(* CODESYS project PFC200_SMS_Alarm.project
   Company: Storm Elektro

Project tree, tasks and I/O mapping:
  PFC200_2ETH_RS_3G : 750-8217 PFC200, WAGO, order no. 750-8217, version 6.1.0.17
    application Application
      libraries: Standard, 3.5.18.0 (System); WagoAppPlcModbus, 1.1.4.8 (WAGO); WagoAppDatalogger, 1.0.5.3 (WAGO); VisuDialogs, * (System); CmpBitmapPool, * (System)
      task Task (cyclic, interval t#50ms, priority 15) calls alarm_test
      task VISU_TASK (cyclic, interval 100 ms, priority 15) calls VisuElems.Visu_Prg
      Symbols
      global variables PersistentVars
      global variables GVL_SMS
      data type DUT_alarm
      text list AlarmListe
      visualisation Visualization
      program alarm_test [ST]: ACT_alarmtekst, ACT_AlarmGruppe, ACT_Alarmliste, ACT_AlarmMottakere, ACT_ReceivdSMS, ACT_SMS_Tjenesten, ACT_ST_SMS_test, ACT_MappingIO
      image pool ImagePool
    Kbus : Kbus, WAGO, version 2.1.0.1
        unmapped channels: K-BUS diagnostics
      XZ200 : 750-1405, WAGO, order no. 750-1405, version 2.0.0.14
          input  xInput1 : BOOL  // _IN._IN
          input  xInput2 : BOOL  // _IN._IN
          input  xInput3 : BOOL  // _IN._IN
          input  xInput4 : BOOL  // _IN._IN
          input  xInput5 : BOOL  // _IN._IN
          input  xInput6 : BOOL  // _IN._IN
          input  xInput7 : BOOL  // _IN._IN
          input  xInput8 : BOOL  // _IN._IN
          input  xInput9 : BOOL  // _IN._IN
          input  xInput10 : BOOL  // _IN._IN
          input  xInput11 : BOOL  // _IN._IN
          input  xInput12 : BOOL  // _IN._IN
          input  xInput13 : BOOL  // _IN._IN
          input  xInput14 : BOOL  // _IN._IN
          input  xInput15 : BOOL  // _IN._IN
          input  xInput16 : BOOL  // _IN._IN
          unmapped channels: _IN
      XZ201 : 750-1405, WAGO, order no. 750-1405, version 2.0.0.14
          input  xInput17 : BOOL  // _IN._IN
          input  xInput18 : BOOL  // _IN._IN
          input  xInput19 : BOOL  // _IN._IN
          input  xInput20 : BOOL  // _IN._IN
          input  xInput21 : BOOL  // _IN._IN
          input  xInput22 : BOOL  // _IN._IN
          input  xInput23 : BOOL  // _IN._IN
          input  xInput24 : BOOL  // _IN._IN
          input  xInput25 : BOOL  // _IN._IN
          input  xInput26 : BOOL  // _IN._IN
          input  xInput27 : BOOL  // _IN._IN
          input  xInput28 : BOOL  // _IN._IN
          input  xInput29 : BOOL  // _IN._IN
          input  xInput30 : BOOL  // _IN._IN
          input  xInput31 : BOOL  // _IN._IN
          input  xInput32 : BOOL  // _IN._IN
          unmapped channels: _IN
      XZ202 : 750-1405, WAGO, order no. 750-1405, version 2.0.0.14
          input  xInput33 : BOOL  // _IN._IN
          input  xInput34 : BOOL  // _IN._IN
          input  xInput35 : BOOL  // _IN._IN
          input  xInput36 : BOOL  // _IN._IN
          input  xInput37 : BOOL  // _IN._IN
          input  xInput38 : BOOL  // _IN._IN
          input  xInput39 : BOOL  // _IN._IN
          input  xInput40 : BOOL  // _IN._IN
          input  xInput41 : BOOL  // _IN._IN
          input  xInput42 : BOOL  // _IN._IN
          input  xInput43 : BOOL  // _IN._IN
          input  xInput44 : BOOL  // _IN._IN
          input  xInput45 : BOOL  // _IN._IN
          input  xInput46 : BOOL  // _IN._IN
          input  xInput47 : BOOL  // _IN._IN
          input  xInput48 : BOOL  // _IN._IN
          unmapped channels: _IN
    Serial
      COM1 : COM1, WAGO, version 0.0.0.19
  libraries: WagoAppSerial_Sms, 1.6.3.2 (WAGO); VisuSymbols, 4.1.0.0 (System); WagoVisuIcons, 1.1.0.5 (WAGO); WagoVisuIconsMaterialDesign, 1.0.0.0 (WAGO)
  text list GlobalTextList
  5ce3da45-db07-42e7-a21c-a00fff4ed8f6|C:\Users\esbo\Downloads\stormlogo.png
*)

// PFC200_2ETH_RS_3G/Application/DUT_alarm
TYPE DUT_alarm :
STRUCT
	TP_Alarm		    : TP;				// Trigger på alarmer
	tTid			    : TIME := T#1S;		// tid
	xAlarm			    : BOOL;				// Alarmgrupper Alarmer som er der nå.
    xAlarm_Trigger      : BOOL;             // Trigger Alarm for å telle antall alarmer
	xIO_input		    : BOOL;				// Input for alarm before timer, enable,disable
	xEnable			    : BOOL := TRUE;		// Enable alarm
	rTrig_Alarm		    : R_TRIG;
	iAlarm_Aktive	    : INT := 0;         // Teller opp antall aktive alarmer
    iAlarm_Ukvitterte	: INT := 0;         // Teller opp antall alarmer siden sist kvittering.
	sAlarmgruppe	    : STRING(255);
	sPrioritet		    : STRING(2);
    xAlarm_GUI          : BOOL;             // alarm til gui
END_STRUCT
END_TYPE

// PFC200_2ETH_RS_3G/Application/PersistentVars
{attribute 'qualified_only'}
VAR_GLOBAL PERSISTENT RETAIN

END_VAR

// PFC200_2ETH_RS_3G/Application/GVL_SMS
{attribute 'qualified_only'}
VAR_GLOBAL
	sAlarmgruppe		: STRING;		// Melding om hvilke alarmgruppe som er utløst
	iAlarmerAktive		: INT := 0;
    iAlarm_Ukvitterte	: INT := 0;         // Teller opp antall alarmer siden sist kvittering.

    xAlarm_GUI          : BOOL;             // alarm til gui
	iAlarmerSendtSMS	: INT := 0;
	iNull				: INT := 0;


	// Trigger SMS sending fra Alarmgruppe, henter det opp i AlarmMottakere 
	xTriggerSms: BOOL;
	// Reseter tellere iAlarmerAktive og iAlarmerSendt
	xKvitter				: BOOL;
	sKvitteringsord			: STRING := 'Kvittert';	//Kvitterings ord
	sKvittering				: STRING := 'Alarmer er kvittert';	//Kvitterings ord
	
	// SMS test
	sSMStest				: STRING := 'Dette er en test av sms sending';	//Kvitterings ord
	xSMStest				: BOOL;	// Test sending av sms
	
END_VAR

VAR_GLOBAL RETAIN
	xNewSmsReceived			: BOOL;
	sMessage				: STRING(GSM_SMS_MSG_MAX_LENGTH);
	// Klargjort for at det skal sendes SMS hvis xTriggerSms og xMobilNR er TRUE
	xMobil_Send				: BOOL;
	xMobil_1_Send			: BOOL;
	xMobil_2_Send			: BOOL;
	xMobil_3_Send			: BOOL;
	iSignalQuality			: INT; 
	xError					: BOOL;    
	oStatus					: WagoSysErrorBase.FbResult;     
	
(*-------------- Melding som skal sendes til SMS Tjeneste ---------------------*)
	xNyMelding				: BOOL := FALSE;
	sNyMelding				: STRING;		// Melding som skal sendes til SMS Tjenesten
	// Alarmvarsel!
	sAlarmVarsel			: STRING(255) := 'Alarm! ' ;
	// AlarmSted
	sAlarmSted				: STRING(255) := 'Alarm place';
	sPrioritet		        : STRING(2);
(*-------------------------------------------------------------------------------------------------------*)
	// Oppdatere mobilNR
	xMobilNR1_CMD			: BOOL := TRUE;
	sMobilNR1				: STRING := '12345678' ;
    xMobilNR1_A_CMD			: BOOL := TRUE;
    xMobilNR1_B_CMD			: BOOL := TRUE; 
    
	xMobilNR2_CMD			: BOOL := TRUE;
	sMobilNR2				: STRING := '87654321' ;
    xMobilNR2_A_CMD			: BOOL := TRUE;
    xMobilNR2_B_CMD			: BOOL := FALSE;     
    
	xMobilNR3_CMD			: BOOL := TRUE;
	sMobilNR3				: STRING := '56784321' ;
    xMobilNR3_A_CMD			: BOOL := TRUE;
    xMobilNR3_B_CMD			: BOOL := TRUE; 
(*--------------Forsinkelse hvis man ikke får kvitterings sms før ny sms sendes---------------------*)
	// Forsinkelsestid
	tAlarmForsinkelse		: TIME := T#24H ;
(*-------------- Pin kode --------------------------------------------------------------------------*)
sPin				: STRING := '9999';	(*pin1: for your sim card like ‘1234’. Empty String means -> no Pin needed*) 

END_VAR

// PFC200_2ETH_RS_3G/Application/alarm_test
PROGRAM alarm_test
VAR
(*----------------------------------------- SMS BLOKK ------------------------------------------------------*)	
(*FbSimpleSms_8207_0	: FbSimpleSms_8207;*)
(*Modem 				: WagoTypesCom.I_WagoSysComBase;*)

my_utSms                 : WagoSysModem.typRxSms;


//xTxInternational	: BOOL;     
my_sTxMessage			: STRING(SMS_CONSTANT.SMS_MSG_MAX_LENGTH) := 'Hello fra SMS_sending' ;			(*(GSM_SMS_MSG_MAX_LENGTH)*) 
my_sTxNumber			: STRING(SMS_CONSTANT.SMS_MSG_MAX_LENGTH) := '12881288';			(*(GSM_PHONE_NO_MAX_LENGTH)*)     
my_receivedMsg          : STRING(SMS_CONSTANT.SMS_MSG_MAX_LENGTH);
my_xTxTriggerSms		: BOOL;				(*start transmission *)
typMy_receivedMsg       : typDeliverSms;
oModemStatus            : WagoSysErrorBase.FbResult;
xSmsSend                : BOOL;				(*TRUE signals that a new message was received -> the application have TO reset THIS variable*) 


GsmMessage              : typGsmMessage;
RxSms                   : typRxSms;
StatusSms               : typStatusSms;
TimeStamp               : typTimeStamp;
UserDataHeader          : typUserDataHeader;

// utTypRxSms 			: wagoappserial_sms.typRxSms;			(*received sms*) 
// eLastSendState		: eErrorGsm;		(*eErrorGsm.OK*)   
//eLastSendStateOK	: eErrorGsm := OK;
// iTxMsgRefNo			: INT; 
(*-------------------------------------------------------------------------------------------------------*)	

	(*--------------Varaibler til FOR LOOP alarmer---------------------*)
	iNull			: INT := 0;
	i				: INT := 0;
	aAlarm			: ARRAY[1..50] OF DUT_alarm;
    iAlarmerAktive_Temp		: INT := 0;
    iAlarm_Ukvitterte_Temp	: INT := 0;         // Teller opp antall alarmer siden sist kvittering.
    
    (*--------------Variabler til GUI------------------------------------*)
	j				: INT := 1;
    k				: INT := 2;
    l				: INT := 3;
    wJ              : WORD := 1;
    dwFillColorAL   : DWORD := 16#FFFF0000;
    dwFrameColorAL   : DWORD := 16#FFFF0000;
    xTest           : BOOL;
    
	(*--------------Forsinkelse hvis man ikke får kvitterings sms før ny sms sendes---------------------*)
	AlarmTimer				: TON;			//Forsinkelse før jeg sender ny alarm
	tAlarmTidCurrent		: TIME;
	xAlarmTidStart			: BOOL;			// Start timer
END_VAR

ACT_alarmtekst();	// Overfører data fra alarm til array

ACT_AlarmGruppe();

ACT_Alarmliste();

ACT_AlarmMottakere();

ACT_SMS_Tjenesten();
ACT_ReceivdSMS();
ACT_ST_SMS_test();
ACT_MappingIO();




//  --- Send SMS
Modem.SmsSend(  sSMSC_No   :='', 
                sDest_No   := my_sTxNumber,
                sMessage   := my_receivedMsg,
                xTxTrigger := my_xTxTriggerSms,
                oStatus    => oModemStatus,
            );


// GUI program
k := j + 1;
l := k + 1;

j := WORD_TO_INT(wJ);

GVL_SMS.xAlarm_GUI := (GVL_SMS.iAlarmerAktive > 0);

ACTION ACT_alarmtekst:
aAlarm[1].sAlarmgruppe := 'B-Alarm Lav temperatur sprinklertank 1';
aAlarm[2].sAlarmgruppe := 'B-Alarm Lav temperatur sprinklertank 2';
aAlarm[3].sAlarmgruppe := 'B-Alarm SM017 ventil stengt';
aAlarm[4].sAlarmgruppe := 'B-Alarm SM015-SM016 ventil stengt';
aAlarm[5].sAlarmgruppe := 'B-Alarm SM010 ventil stengt';
aAlarm[6].sAlarmgruppe := 'B-Alarm SM013-SM014 ventil stengt';
aAlarm[7].sAlarmgruppe := 'B-Alarm SM019 ventil stengt';
aAlarm[8].sAlarmgruppe := 'B-Alarm SM021 ventil stengt'; 
aAlarm[9].sAlarmgruppe := 'B-Alarm SM022 ventil stengt';
aAlarm[10].sAlarmgruppe := 'B-Alarm SM023 ventil stengt';
aAlarm[11].sAlarmgruppe := 'B-Alarm SM024 ventil stengt';
aAlarm[12].sAlarmgruppe := 'B-Alarm SM003-SM004 ventil stengt';
aAlarm[13].sAlarmgruppe := 'B-Alarm QP001 lavt trykk kommunal ledning';
aAlarm[14].sAlarmgruppe := 'B-Alarm SM001-SM002 ventil stengt';
aAlarm[15].sAlarmgruppe := 'B-Alarm SM025 ventil stengt';
aAlarm[16].sAlarmgruppe := 'B-Alarm RT001 lav temperatur pumperom';

aAlarm[17].sAlarmgruppe := 'B-Alarm Sprinklerpumpe 1 - i drift';
aAlarm[18].sAlarmgruppe := 'B-Alarm Sprinklerpumpe 1 - Motor alarm';
aAlarm[19].sAlarmgruppe := 'B-Alarm Sprinklerpumpe 1 - Automatikk alarm';
aAlarm[20].sAlarmgruppe := 'B-Alarm Sprinklerpumpe 1 – Pumperom alarm';
aAlarm[21].sAlarmgruppe := 'B-Alarm Sprinklerpumpe 1 – Ikke i Auto';
aAlarm[22].sAlarmgruppe := 'B-Alarm SM012 ventil stengt';
aAlarm[23].sAlarmgruppe := 'B-Alarm RN003 Lavt nivå sprinklertank 1';
aAlarm[24].sAlarmgruppe := 'B-Alarm RN004 Høy nivå sprinklertank 1';
aAlarm[25].sAlarmgruppe := 'B-Alarm Sprinklerpumpe 2 - i drift';
aAlarm[26].sAlarmgruppe := 'B-Alarm Sprinklerpumpe 2 - Motor alarm';
aAlarm[27].sAlarmgruppe := 'B-Alarm Sprinklerpumpe 2 - Automatikk alarm';
aAlarm[28].sAlarmgruppe := 'B-Alarm Sprinklerpumpe 2 – Pumperom alarm';
aAlarm[29].sAlarmgruppe := 'B-Alarm Sprinklerpumpe 2 – Ikke i Auto';
aAlarm[30].sAlarmgruppe := 'B-Alarm RN005 Lavt nivå sprinklertank 2';
aAlarm[31].sAlarmgruppe := 'A-Alarm RN006 Høy nivå sprinklertank 2';
aAlarm[32].sAlarmgruppe := 'Ledig';
aAlarm[33].sAlarmgruppe := 'A-Alarm Sprinkler utløst pumperom';
aAlarm[34].sAlarmgruppe := 'A-Alarm Sprinklerpumpe 1 i drift';
aAlarm[35].sAlarmgruppe := 'A-Alarm Sprinklerpumpe 2 i drift';

aAlarm[1].sPrioritet := 'B';
aAlarm[2].sPrioritet := 'B';
aAlarm[3].sPrioritet := 'B';
aAlarm[4].sPrioritet := 'B';
aAlarm[5].sPrioritet := 'B';
aAlarm[6].sPrioritet := 'B';
aAlarm[7].sPrioritet := 'B';
aAlarm[8].sPrioritet := 'B';
aAlarm[9].sPrioritet := 'B';
aAlarm[10].sPrioritet := 'B';
aAlarm[11].sPrioritet := 'B';
aAlarm[12].sPrioritet := 'B';
aAlarm[13].sPrioritet := 'B';
aAlarm[14].sPrioritet := 'B';
aAlarm[15].sPrioritet := 'B';
aAlarm[16].sPrioritet := 'B';
aAlarm[17].sPrioritet := 'B';
aAlarm[18].sPrioritet := 'B';
aAlarm[19].sPrioritet := 'B';
aAlarm[20].sPrioritet := 'B';
aAlarm[21].sPrioritet := 'B';
aAlarm[22].sPrioritet := 'B';
aAlarm[23].sPrioritet := 'B';
aAlarm[24].sPrioritet := 'B';
aAlarm[25].sPrioritet := 'B';
aAlarm[26].sPrioritet := 'B';
aAlarm[27].sPrioritet := 'B';
aAlarm[28].sPrioritet := 'B';
aAlarm[29].sPrioritet := 'B';
aAlarm[30].sPrioritet := 'B';
aAlarm[31].sPrioritet := 'A';
aAlarm[33].sPrioritet := '';
aAlarm[33].sPrioritet := 'A';
aAlarm[34].sPrioritet := 'A';
aAlarm[35].sPrioritet := 'A';
END_ACTION

ACTION ACT_AlarmGruppe:
FOR i := 1 TO 40 DO
  aAlarm[i].rTrig_Alarm(CLK := aAlarm[i].xAlarm);
  aAlarm[i].xAlarm_GUI := (aAlarm[i].iAlarm_Ukvitterte > 0);
    IF aAlarm[i].rTrig_Alarm.Q = TRUE THEN
		aAlarm[i].iAlarm_Ukvitterte := aAlarm[i].iAlarm_Ukvitterte +1;
        wJ := INT_TO_WORD(i);
        GVL_SMS.iAlarm_Ukvitterte := GVL_SMS.iAlarm_Ukvitterte + 1;
		GVL_SMS.sAlarmgruppe := aAlarm[i].sAlarmgruppe;
        GVL_SMS.sPrioritet  := aAlarm[i].sPrioritet; 
    END_IF
END_FOR

IF GVL_SMS.iAlarm_Ukvitterte > GVL_SMS.iNull THEN
    AlarmTimer(IN := xAlarmTidStart, PT := GVL_SMS.tAlarmForsinkelse);
    xAlarmTidStart := TRUE;
    tAlarmTidCurrent := AlarmTimer.ET;
    IF AlarmTimer.Q = TRUE THEN
        GVL_SMS.xTriggerSms := TRUE;
        xAlarmTidStart := FALSE;
    END_IF
ELSE
    xAlarmTidStart := FALSE;
END_IF

IF GVL_SMS.xKvitter = TRUE THEN
    FOR i := 1 TO 40 DO
        aAlarm[i].iAlarm_Ukvitterte := 0;
    END_FOR
    GVL_SMS.iAlarm_Ukvitterte := 0;
    GVL_SMS.iAlarmerSendtSMS := 0;
    GVL_SMS.sAlarmgruppe := GVL_SMS.sKvittering;
    GVL_SMS.xTriggerSms := TRUE;
    GVL_SMS.xKvitter := FALSE;
    GVL_SMS.sPrioritet  := '';
END_IF


IF (GVL_SMS.iAlarm_Ukvitterte > GVL_SMS.iNull) AND (GVL_SMS.iAlarmerSendtSMS < GVL_SMS.iAlarm_Ukvitterte) THEN

	GVL_SMS.xTriggerSms := TRUE;
	GVL_SMS.iAlarmerSendtSMS := GVL_SMS.iAlarmerSendtSMS +1;
END_IF


IF (GVL_SMS.iAlarm_Ukvitterte > GVL_SMS.iNull) THEN
	AlarmTimer(IN := xAlarmTidStart, PT:= GVL_SMS.tAlarmForsinkelse);
			xAlarmTidStart := TRUE;
			tAlarmTidCurrent := AlarmTimer.ET;
				IF AlarmTimer.Q = TRUE THEN
					GVL_SMS.xTriggerSms := TRUE;
					xAlarmTidStart := FALSE;
				END_IF
ELSE 
	xAlarmTidStart := FALSE;
END_IF
END_ACTION

ACTION ACT_Alarmliste:

// Tar input IO, sjekker om den er TRUE, Forsinkelse Før alarmen går videre. Må enable alarmen.
// Alarm innganger er da aAlarm[1].xIO_input og aAlarm[2].xIO_input osv
FOR i := 1 TO 40 DO
	aAlarm[i].TP_Alarm(	IN:=aAlarm[i].xIO_input,
						PT:=aAlarm[i].tTid,
						Q=>,
						ET=> 
						);
	aAlarm[i].xAlarm_Trigger	:= aAlarm[i].xEnable AND aAlarm[i].TP_Alarm.Q;
END_FOR


    iAlarmerAktive_Temp		:= 0;
    iAlarm_Ukvitterte_Temp	:= 0;    
    FOR i := 1 TO 40 DO
	    aAlarm[i].xAlarm	        := aAlarm[i].xIO_input;
        iAlarm_Ukvitterte_Temp   := iAlarm_Ukvitterte_Temp + aAlarm[i].iAlarm_Ukvitterte;
        IF aAlarm[i].xAlarm = TRUE THEN
            iAlarmerAktive_Temp      := iAlarmerAktive_Temp + 1;
        END_IF 
    END_FOR
    
GVL_SMS.iAlarmerAktive := iAlarmerAktive_Temp;
GVL_SMS.iAlarm_Ukvitterte := iAlarm_Ukvitterte_Temp;
END_ACTION

ACTION ACT_AlarmMottakere:
IF (GVL_SMS.xTriggerSms = TRUE) THEN
	GVL_SMS.xMobil_Send		:= TRUE;
	GVL_SMS.xMobil_1_Send	:= GVL_SMS.xMobilNR1_CMD;
	GVL_SMS.xMobil_2_Send	:= GVL_SMS.xMobilNR2_CMD;
	GVL_SMS.xMobil_3_Send	:= GVL_SMS.xMobilNR3_CMD;
	GVL_SMS.xTriggerSms 	:= FALSE;
END_IF
	 
IF (GVL_SMS.xMobil_1_Send = TRUE) AND (my_xTxTriggerSms = FALSE) THEN
    IF GVL_SMS.xMobilNR1_A_CMD = TRUE AND GVL_SMS.sPrioritet = 'A' THEN
		my_sTxNumber := GVL_SMS.sMobilNR1;
		my_xTxTriggerSms := TRUE;	// Sende SMS
		GVL_SMS.xMobil_1_Send := FALSE;
    END_IF
    IF GVL_SMS.xMobilNR1_B_CMD = TRUE AND GVL_SMS.sPrioritet = 'B' THEN
		my_sTxNumber := GVL_SMS.sMobilNR1;
		my_xTxTriggerSms := TRUE;	// Sende SMS
		GVL_SMS.xMobil_1_Send := FALSE;
    END_IF    
END_IF
	

IF (GVL_SMS.xMobil_2_Send = TRUE) AND (my_xTxTriggerSms = FALSE) THEN
    IF GVL_SMS.xMobilNR2_A_CMD = TRUE AND GVL_SMS.sPrioritet = 'A' THEN
		my_sTxNumber := GVL_SMS.sMobilNR2;
		my_xTxTriggerSms := TRUE;	// Sende SMS
		GVL_SMS.xMobil_2_Send := FALSE;
    END_IF
    IF GVL_SMS.xMobilNR2_B_CMD = TRUE AND GVL_SMS.sPrioritet = 'B' THEN
		my_sTxNumber := GVL_SMS.sMobilNR2;
		my_xTxTriggerSms := TRUE;	// Sende SMS
		GVL_SMS.xMobil_2_Send := FALSE;
    END_IF    
END_IF

IF (GVL_SMS.xMobil_3_Send = TRUE) AND (my_xTxTriggerSms = FALSE) THEN
    IF GVL_SMS.xMobilNR3_A_CMD = TRUE AND GVL_SMS.sPrioritet = 'A' THEN
		my_sTxNumber := GVL_SMS.sMobilNR3;
		my_xTxTriggerSms := TRUE;	// Sende SMS
		GVL_SMS.xMobil_3_Send := FALSE;
    END_IF
    IF GVL_SMS.xMobilNR3_B_CMD = TRUE AND GVL_SMS.sPrioritet = 'B' THEN
		my_sTxNumber := GVL_SMS.sMobilNR3;
		my_xTxTriggerSms := TRUE;	// Sende SMS
		GVL_SMS.xMobil_3_Send := FALSE;
    END_IF
END_IF


IF (GVL_SMS.xTriggerSms = TRUE) AND (GVL_SMS.xMobil_1_Send = FALSE) AND (GVL_SMS.xMobil_2_Send = FALSE) AND (GVL_SMS.xMobil_3_Send = FALSE) THEN
	GVL_SMS.xTriggerSms := FALSE;
END_IF
	
IF (GVL_SMS.xMobil_Send	= TRUE) AND (GVL_SMS.xMobil_1_Send = FALSE) AND (GVL_SMS.xMobil_2_Send = FALSE) AND (GVL_SMS.xMobil_3_Send = FALSE) THEN
	GVL_SMS.xMobil_Send	:= FALSE;
END_IF
END_ACTION

ACTION ACT_ReceivdSMS:

//--- RECEIVE SMS ----------------------------------------------------------------
IF Modem.SmsReceive(my_utSms) THEN // a new message was received	
	// process here the new message
	my_receivedMsg := my_utSms.DeliverSms.Msg;
    GVL_SMS.sMessage := my_utSms.DeliverSms.Msg;
    IF GVL_SMS.sKvitteringsord  = my_receivedMsg THEN
	    GVL_SMS.xKvitter := TRUE;
	END_IF 
	
END_IF
//--------------------------------------------------------------------------------
END_ACTION

ACTION ACT_SMS_Tjenesten:
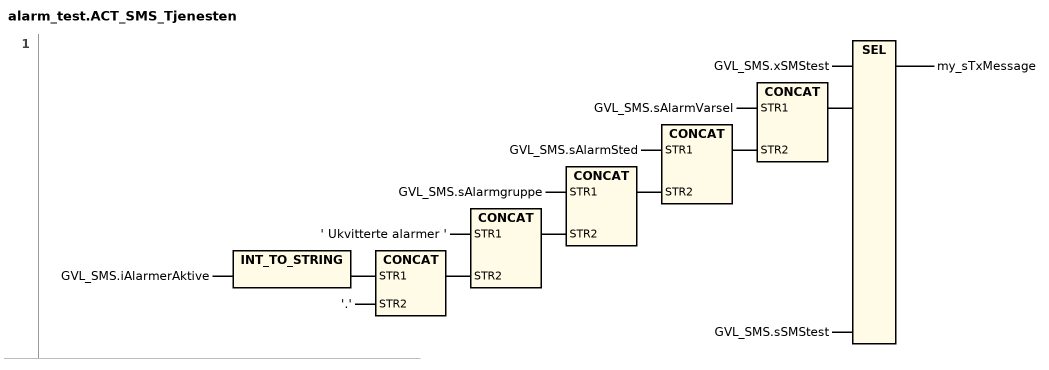
// NETWORK 1
my_sTxMessage := SEL(GVL_SMS.xSMStest, CONCAT(STR1 := GVL_SMS.sAlarmVarsel, STR2 := CONCAT(STR1 := GVL_SMS.sAlarmSted, STR2 := CONCAT(STR1 := GVL_SMS.sAlarmgruppe, STR2 := CONCAT(STR1 := ' Ukvitterte alarmer ', STR2 := CONCAT(STR1 := INT_TO_STRING(GVL_SMS.iAlarmerAktive), STR2 := '.'))))), GVL_SMS.sSMStest);
END_ACTION

ACTION ACT_ST_SMS_test:
IF (GVL_SMS.xSMStest = TRUE) THEN
	GVL_SMS.xMobil_Send		:= TRUE;
	GVL_SMS.xMobil_1_Send	:= GVL_SMS.xMobilNR1_CMD;
	GVL_SMS.xMobil_2_Send	:= GVL_SMS.xMobilNR2_CMD;
	GVL_SMS.xMobil_3_Send	:= GVL_SMS.xMobilNR3_CMD;
	GVL_SMS.xTriggerSms 	:= FALSE;
END_IF
	 
IF (GVL_SMS.xMobil_1_Send = TRUE) AND (my_xTxTriggerSms = FALSE) THEN
		my_sTxNumber := GVL_SMS.sMobilNR1;
		my_sTxMessage := GVL_SMS.sSMStest;
		my_xTxTriggerSms := TRUE;	// Sende SMS
		GVL_SMS.xMobil_1_Send := FALSE;
END_IF
	

IF (GVL_SMS.xMobil_2_Send = TRUE) AND (my_xTxTriggerSms = FALSE) THEN
	my_sTxNumber := GVL_SMS.sMobilNR2;
	my_sTxMessage := GVL_SMS.sSMStest;
	my_xTxTriggerSms := TRUE;	// Sende SMS
	GVL_SMS.xMobil_2_Send := FALSE; 
END_IF

IF (GVL_SMS.xMobil_3_Send = TRUE) AND (my_xTxTriggerSms = FALSE) THEN
	my_sTxNumber := GVL_SMS.sMobilNR3;
	my_sTxMessage := GVL_SMS.sSMStest;
	my_xTxTriggerSms := TRUE;	// Sende SMS
	GVL_SMS.xMobil_3_Send := FALSE; 
END_IF


IF (GVL_SMS.xTriggerSms = TRUE) AND (GVL_SMS.xMobil_1_Send = FALSE) AND (GVL_SMS.xMobil_2_Send = FALSE) AND (GVL_SMS.xMobil_3_Send = FALSE) THEN
	GVL_SMS.xTriggerSms := FALSE;
END_IF
	
IF (GVL_SMS.xMobil_Send	= TRUE) AND (GVL_SMS.xMobil_1_Send = FALSE) AND (GVL_SMS.xMobil_2_Send = FALSE) AND (GVL_SMS.xMobil_3_Send = FALSE) THEN
	GVL_SMS.xMobil_Send	:= FALSE;
END_IF
END_ACTION

ACTION ACT_MappingIO:

alarm_test.aAlarm[1].xIO_input := xInput1;
alarm_test.aAlarm[2].xIO_input := xInput2;
alarm_test.aAlarm[3].xIO_input := xInput3;
alarm_test.aAlarm[4].xIO_input := xInput4;
alarm_test.aAlarm[5].xIO_input := xInput5;
alarm_test.aAlarm[6].xIO_input := xInput6;
alarm_test.aAlarm[7].xIO_input := xInput7;
alarm_test.aAlarm[8].xIO_input := xInput8;
alarm_test.aAlarm[9].xIO_input := xInput9;
alarm_test.aAlarm[10].xIO_input := xInput10;
alarm_test.aAlarm[11].xIO_input := xInput11;
alarm_test.aAlarm[12].xIO_input := xInput12;
alarm_test.aAlarm[13].xIO_input := xInput13;
alarm_test.aAlarm[14].xIO_input := xInput14;
alarm_test.aAlarm[15].xIO_input := xInput15;
alarm_test.aAlarm[16].xIO_input := xInput16;
alarm_test.aAlarm[17].xIO_input := xInput17;
alarm_test.aAlarm[18].xIO_input := xInput18;
alarm_test.aAlarm[19].xIO_input := xInput19;
alarm_test.aAlarm[20].xIO_input := xInput20;
alarm_test.aAlarm[21].xIO_input := xInput21;
alarm_test.aAlarm[22].xIO_input := xInput22;
alarm_test.aAlarm[23].xIO_input := xInput23;
alarm_test.aAlarm[24].xIO_input := xInput24;
alarm_test.aAlarm[25].xIO_input := xInput25;
alarm_test.aAlarm[26].xIO_input := xInput26;
alarm_test.aAlarm[27].xIO_input := xInput27;
alarm_test.aAlarm[28].xIO_input := xInput28;
alarm_test.aAlarm[29].xIO_input := xInput29;
alarm_test.aAlarm[30].xIO_input := xInput30;
alarm_test.aAlarm[31].xIO_input := xInput31;
alarm_test.aAlarm[32].xIO_input := xInput32;
alarm_test.aAlarm[33].xIO_input := xInput33;
alarm_test.aAlarm[34].xIO_input := xInput34;
alarm_test.aAlarm[35].xIO_input := xInput35;
alarm_test.aAlarm[36].xIO_input := xInput36;
alarm_test.aAlarm[37].xIO_input := xInput37;
alarm_test.aAlarm[38].xIO_input := xInput38;
alarm_test.aAlarm[39].xIO_input := xInput39;
alarm_test.aAlarm[40].xIO_input := xInput40;
alarm_test.aAlarm[41].xIO_input := xInput41;
alarm_test.aAlarm[42].xIO_input := xInput42;
alarm_test.aAlarm[43].xIO_input := xInput43;
alarm_test.aAlarm[44].xIO_input := xInput44;
alarm_test.aAlarm[45].xIO_input := xInput45;
alarm_test.aAlarm[46].xIO_input := xInput46;
alarm_test.aAlarm[47].xIO_input := xInput47;
alarm_test.aAlarm[48].xIO_input := xInput48;
END_ACTION

END_PROGRAM

// PFC200_2ETH_RS_3G/Application/Visualization
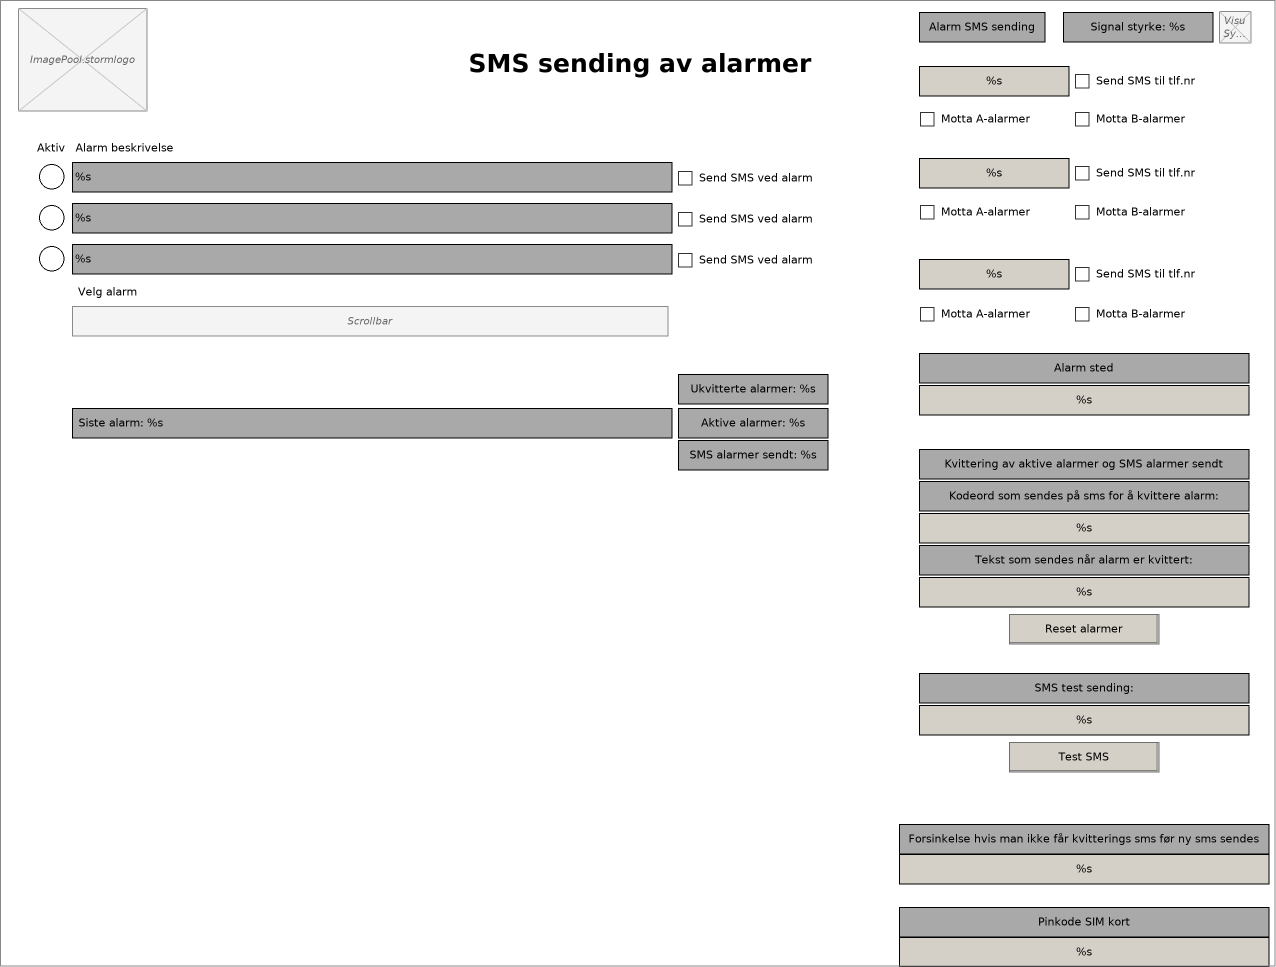
VISUALIZATION Visualization  // 1276x967
    Rectangle (919,449 330x30), "Kvittering av aktive alarmer og SMS alarmer sendt"
    Rectangle (919,66 150x30), "%s", text variable: GVL_SMS.sMobilNR1
        OnMouseClick: write the text variable via Default
    Rectangle (72,162 600x30), "%s", tooltip "Alarm beskrivelse", text variable: alarm_test.aAlarm[alarm_test.j].sAlarmgruppe, colour toggle: alarm_test.aAlarm[alarm_test.j].xAlarm_GUI
    Checkbox (676,163 150x30), "Send SMS ved alarm", variable: alarm_test.aAlarm[alarm_test.j].xEnable
    Checkbox (1073,66 150x30), "Send SMS til tlf.nr", variable: GVL_SMS.xMobilNR1_CMD
    Rectangle (919,158 150x30), "%s", text variable: GVL_SMS.sMobilNR2
        OnMouseClick: write the text variable via Default
    Checkbox (1073,158 150x30), "Send SMS til tlf.nr", variable: GVL_SMS.xMobilNR2_CMD
    Rectangle (919,259 150x30), "%s", text variable: GVL_SMS.sMobilNR3
        OnMouseClick: write the text variable via Default
    Checkbox (1073,259 150x30), "Send SMS til tlf.nr", variable: GVL_SMS.xMobilNR3_CMD
    Rectangle (72,408 600x30), "Siste alarm: %s", text variable: GVL_SMS.sAlarmgruppe, colour toggle: GVL_SMS.xAlarm_GUI
    Rectangle (678,408 150x30), "Aktive alarmer: %s", text variable: GVL_SMS.iAlarmerAktive
    Rectangle (678,440 150x30), "SMS alarmer sendt: %s", text variable: GVL_SMS.iAlarmerSendtSMS
    Button (1009,614 150x30), "Reset alarmer"
        tap GVL_SMS.xKvitter
    Rectangle (919,513 330x30), "%s", text variable: GVL_SMS.sKvitteringsord
        OnMouseClick: write the text variable via Default
    Rectangle (919,481 330x30), "Kodeord som sendes på sms for å kvittere alarm:"
    Rectangle (919,545 330x30), "Tekst som sendes når alarm er kvittert:"
    Rectangle (919,577 330x30), "%s", text variable: GVL_SMS.sKvittering
        OnMouseClick: write the text variable via Default
    Button (1009,742 150x30), "Test SMS"
        tap GVL_SMS.xSMStest
    Rectangle (919,673 330x30), "SMS test sending:"
    Rectangle (919,705 330x30), "%s", text variable: GVL_SMS.sSMStest
        OnMouseClick: write the text variable via Default
    Image (1219,11 32x32), image: VisuSymbols.Symbols.Signal
    Rectangle (1063,12 150x30), "Signal styrke: %s", text variable: GVL_SMS.iSignalQuality
    Rectangle (919,12 126x30), "Alarm SMS sending", colour toggle: GVL_SMS.xError
    Rectangle (919,353 330x30), "Alarm sted"
    Rectangle (919,385 330x30), "%s", text variable: GVL_SMS.sAlarmSted
        OnMouseClick: write the text variable via Default
    Rectangle (899,854 370x30), "%s", text variable: GVL_SMS.tAlarmForsinkelse
        OnMouseClick: write the text variable via Default
    Rectangle (899,824 370x30), "Forsinkelse hvis man ikke får kvitterings sms før ny sms sendes"
    Rectangle (899,907 370x30), "Pinkode SIM kort"
    Rectangle (899,937 370x30), "%s", text variable: GVL_SMS.sPin
        OnMouseClick: write the text variable via Default
    Label (4,48 1272x30), "SMS sending av alarmer"
    Rectangle (72,203 600x30), "%s", tooltip "Alarm beskrivelse", text variable: alarm_test.aAlarm[alarm_test.k].sAlarmgruppe, colour toggle: alarm_test.aAlarm[alarm_test.k].xAlarm_GUI
    Checkbox (676,204 150x30), "Send SMS ved alarm", variable: alarm_test.aAlarm[alarm_test.k].xEnable
    Rectangle (72,244 600x30), "%s", tooltip "Alarm beskrivelse", text variable: alarm_test.aAlarm[alarm_test.l].sAlarmgruppe, colour toggle: alarm_test.aAlarm[alarm_test.l].xAlarm_GUI
    Checkbox (676,245 150x30), "Send SMS ved alarm", variable: alarm_test.aAlarm[alarm_test.l].xEnable
    Scrollbar (72,306 596x30)
        p1057716461: alarm_test.wJ
    Image (18,8 129x103), image: ImagePool.stormlogo
    Ellipse (39,164 25x25), tooltip "Fysisk alarm", colour toggle: alarm_test.aAlarm[alarm_test.j].xAlarm
    Ellipse (39,205 25x25), tooltip "Fysisk alarm", colour toggle: alarm_test.aAlarm[alarm_test.k].xAlarm
    Ellipse (39,246 25x25), tooltip "Fysisk alarm", colour toggle: alarm_test.aAlarm[alarm_test.l].xAlarm
    Label (33,136 36x24), "Aktiv"
    Label (72,136 105x24), "Alarm beskrivelse"
    Label (72,280 71x24), "Velg alarm"
    Rectangle (678,374 150x30), "Ukvitterte alarmer: %s", text variable: GVL_SMS.iAlarm_Ukvitterte
    Checkbox (1073,104 150x30), "Motta B-alarmer", variable: GVL_SMS.xMobilNR1_B_CMD
    Checkbox (918,104 150x30), "Motta A-alarmer", variable: GVL_SMS.xMobilNR1_A_CMD
    Checkbox (918,197 150x30), "Motta A-alarmer", variable: GVL_SMS.xMobilNR2_A_CMD
    Checkbox (1073,197 150x30), "Motta B-alarmer", variable: GVL_SMS.xMobilNR2_B_CMD
    Checkbox (918,299 150x30), "Motta A-alarmer", variable: GVL_SMS.xMobilNR3_A_CMD
    Checkbox (1073,299 150x30), "Motta B-alarmer", variable: GVL_SMS.xMobilNR3_B_CMD
END_VISUALIZATION

(* text list AlarmListe (id | default)
  AL_1 | 
   |  *)
